FUNCTION_BLOCK SRSection
  (* Standard: 61499-2 *)
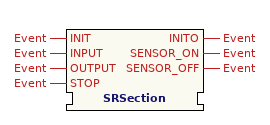
  EVENT_INPUT
    INIT;
    INPUT;
    OUTPUT;
    STOP;
  END_EVENT
  EVENT_OUTPUT
    INITO;
    SENSOR_ON;
    SENSOR_OFF;
  END_EVENT
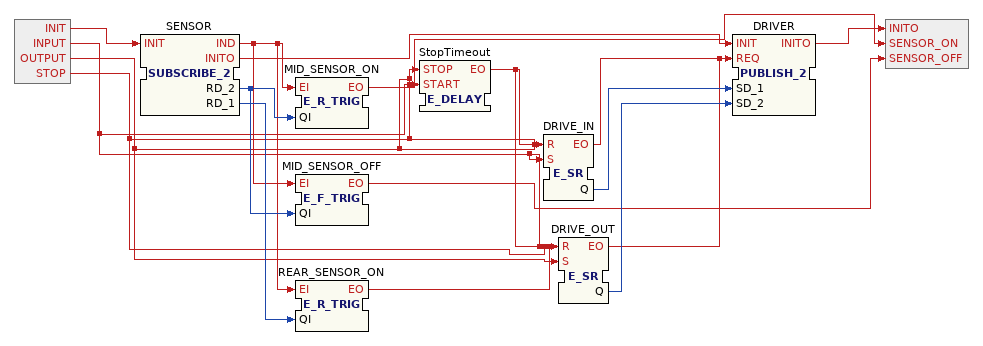
  FBS
    DRIVER : PUBLISH_2;
    SENSOR : SUBSCRIBE_2;
    DRIVE_IN : E_SR;
    MID_SENSOR_ON : E_R_TRIG;
    MID_SENSOR_OFF : E_F_TRIG;
    StopTimeout : E_DELAY;
    DRIVE_OUT : E_SR;
    REAR_SENSOR_ON : E_R_TRIG;
  END_FBS
  EVENT_CONNECTIONS
    MID_SENSOR_ON.EO TO SENSOR_ON;
    MID_SENSOR_OFF.EO TO SENSOR_OFF;
    StopTimeout.EO TO DRIVE_IN.R;
    INIT TO SENSOR.INIT;
    SENSOR.IND TO MID_SENSOR_ON.EI;
    SENSOR.IND TO MID_SENSOR_OFF.EI;
    SENSOR.INITO TO DRIVER.INIT;
    DRIVE_IN.EO TO DRIVER.REQ;
    DRIVER.INITO TO INITO;
    DRIVE_OUT.EO TO DRIVER.REQ;
    StopTimeout.EO TO DRIVE_OUT.R;
    INPUT TO DRIVE_IN.S;
    OUTPUT TO DRIVE_OUT.S;
    STOP TO DRIVE_IN.R;
    STOP TO StopTimeout.STOP;
    STOP TO DRIVE_OUT.R;
    OUTPUT TO DRIVE_IN.R;
    INPUT TO DRIVE_OUT.R;
    INPUT TO StopTimeout.START;
    OUTPUT TO StopTimeout.START;
    SENSOR.IND TO REAR_SENSOR_ON.EI;
    REAR_SENSOR_ON.EO TO DRIVE_OUT.R;
  END_CONNECTIONS
  DATA_CONNECTIONS
    SENSOR.RD_2 TO MID_SENSOR_ON.QI;
    SENSOR.RD_2 TO MID_SENSOR_OFF.QI;
    DRIVE_IN.Q TO DRIVER.SD_1;
    DRIVE_OUT.Q TO DRIVER.SD_2;
    SENSOR.RD_1 TO REAR_SENSOR_ON.QI;
  END_CONNECTIONS
END_FUNCTION_BLOCK
